FUNCTION c_to_f : REAL
VAR_INPUT
	tempC : REAL;
END_VAR
VAR
END_VAR

c_to_f := (tempC*1.8) + 32;

END_FUNCTION

(* stored: Version 1.1.0.1, ProductVersion 3.1.4024.12
   POU c_to_f: Id {a4b81a62-9f9e-4bc0-b40c-689fff09d50f}, SpecialFunc None *)
